# EPICS autosave request: iocBoot/sioc-asta-stats02/pvStats.req
file ../pvStatsCommon.req P=$(P)
file ../pvStatsScope.req P=$(P)
